TYPE ST_BuzzCtrl :
STRUCT
	Command : ST_CommandBasic;
	Status	: ST_StatusBasic;
	BuzzTime	: LREAL;
END_STRUCT
END_TYPE

(* stored: Version 1.1.0.1, ProductVersion 3.1.4024.13
   DUT ST_BuzzCtrl: Id {ef602a1e-786b-4d32-88db-2df5e068a955} *)
